ABB RobotStudio station: Lab1_5_20210903-135838.rsstn

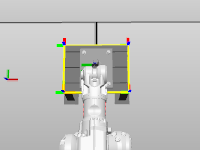
Station Lab1_4 (saved by RobotStudio 21.2.9526.0)
Layout (positions relative to the parent item):
  - IRB140_6_81_C_03 [mechanism, from Robots\IRB140_6_81_C_G_03.rslib] at (0, 0, 0) mm; joint values [0, 0, 0.1367, 0.0158, 0.861, 0] (rad or m)
  - UISpenholder [mechanism, from RS1\UISpenholder.rslib] at (481.7, 0.78, 605.59) mm, rotated rx 178.93 ry 32.83 rz 179.3 deg
  - table_and_fixture_140 [part, from Training Objects\propeller_table.rslib] at (400, 220, 0) mm, rotated rx 0 ry 0 rz -90 deg
Attachment: UISpenholder is attached to IRB140_6_81_C_03 / Link6
Attachment: WobjTable is attached to table_and_fixture_140
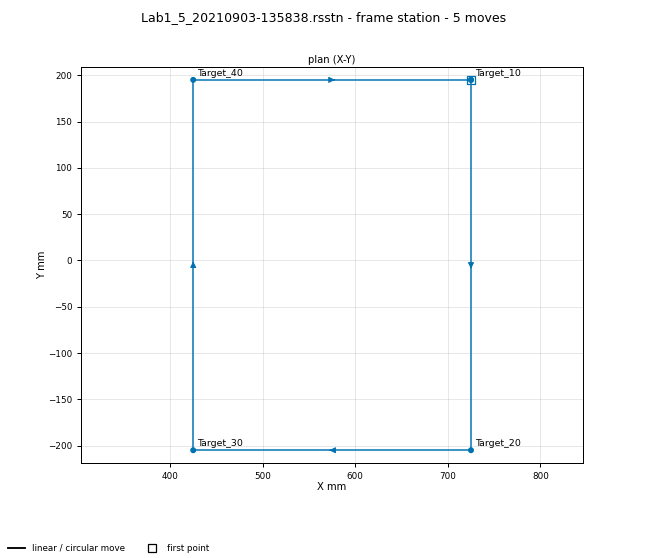
[picture p0: tool path of Lab1_5_20210903-135838.rsstn in frame station, 5 of 5 moves have a stored position in this frame; points joined in program order, loops and branches not executed]
Targets, tools, work objects and paths stored in the station, written as RAPID:
! task (no controller)
MODULE CalibData
  TASK PERS wobjdata WobjTable:=[FALSE,TRUE,"",[[575,620,0],[0.707106781,0,0,-0.707106781]],[[425,-150,308],[1,0,0,0]]];
ENDMODULE

! task (no controller)
MODULE Module1
  CONST robtarget Target_10:=[[0,300,0],[0.707106781,0,0,0.707106781],[0,0,0,0],[9E+09,9E+09,9E+09,9E+09,9E+09,9E+09]];
  CONST robtarget Target_20:=[[400,300,0],[0.707106781,0,0,0.707106781],[0,0,0,0],[9E+09,9E+09,9E+09,9E+09,9E+09,9E+09]];
  CONST robtarget Target_30:=[[400,0,0],[0.707106781,0,0,0.707106781],[0,0,0,0],[9E+09,9E+09,9E+09,9E+09,9E+09,9E+09]];
  CONST robtarget Target_40:=[[0,0,0],[0.707106781,0,0,0.707106781],[0,0,0,0],[9E+09,9E+09,9E+09,9E+09,9E+09,9E+09]];
  PROC Path_10()
    MoveL Target_10,v1000,z5,tool0\WObj:=WobjTable;
    MoveL Target_20,v1000,z5,tool0\WObj:=WobjTable;
    MoveL Target_30,v1000,z5,tool0\WObj:=WobjTable;
    MoveL Target_40,v1000,z5,tool0\WObj:=WobjTable;
    MoveL Target_10,v1000,z5,tool0\WObj:=WobjTable;
  ENDPROC
ENDMODULE

! task (no controller)
MODULE CalibData
  PERS tooldata UISpenholder:=[TRUE,[[0,0,110],[1,0,0,0]],[1,[0,0,1],[1,0,0,0],0,0,0]];
ENDMODULE

